TYPE ST_DriveAlarmCode :
STRUCT
	Error1	: USINT;
	Error2	: USINT;
	Error3	: USINT;
	Error4	: USINT;
END_STRUCT
END_TYPE

(* stored: Version 1.1.0.1, ProductVersion 3.1.4024.9
   DUT ST_DriveAlarmCode: Id {61ca4a1d-8bec-434a-baa7-1a391c8244f9} *)
